TYPE ST_StepStatus :
STRUCT
 xStart:BOOL;
 xBusy:BOOL;
 xDone:BOOL;
 xError:BOOL;
END_STRUCT
END_TYPE

(* stored: Version 1.1.0.1, ProductVersion 3.1.4024.9
   DUT ST_StepStatus: Id {9be2ccf8-2bad-4700-a045-63ea4d161403} *)
